FUNCTION_BLOCK A2X_PUBLISH_2 (* Publish both BOOLs of an A2X adapter to one or many SUBSCRIBE_2 Blocks, each buffered with an E_D_FF. Contract: garantiert seit v1.1 einen erzwungenen ersten Publish direkt nach INIT (OPC-UA-Knoten existiert sofort, auch ohne vorherige echte Wertaenderung am Adapter) - dieser erste Publish kann aber noch den Default-/Platzhalterwert des internen Latches enthalten statt des tatsaechlichen aktuellen Adapterwerts, bis die erste echte Aenderung eintrifft. Consumer, die auf den exakten Erstwert angewiesen sind, muessen das beruecksichtigen. Verhalten bei QI=FALSE (deaktivierter Publisher) verifiziert (FORTE-Quellcode, core/src/cominfra/commfb.cpp): weder beim INIT (Verbindung wird geschlossen statt geoeffnet) noch beim erzwungenen Erst-Publish (sendData() bricht vor dem Erreichen der Kommunikationsschicht ab) wird tatsaechlich etwas gesendet oder ein Knoten angelegt - das dabei ausgeloeste CNF/QO=FALSE/STATUS=Inhibited ist reine lokale Rueckmeldung, keine Netzwerkoperation, unbedenklich. Ein spaeterer QI-Wechsel FALSE->TRUE ohne erneutes INIT loest den erzwungenen Erst-Publish NICHT erneut aus. *)
  (* Standard: 61499-2; Description: Copyright (c) 2026 HR Agrartechnik GmbH This program and the accompanying materials are made available under the terms of the Eclipse Public License 2.0 which is available at https://www.eclipse.org/legal/epl-2.0/ SPDX-License-Identifier: EPL-2.0 *)
  (* Version 1.1, 2026-09-17, Franz Höpfinger, HR Agrartechnik GmbH, Erzwungener Erst-Publish nach INIT: PUBLISH_1/PUBLISH_2.INITO -> .REQ ergaenzt (Franz, gegen fehlende OPC-UA-Knoten wenn seit Power-On noch keine echte Wertaenderung stattfand, siehe BERICHT_2026-09-16_STG3_I1_I3_I4_I6_STALE_REMOTE_SUBSCRIBE.md Abschnitt 18-20) - garantiert einen unbedingten ersten Publish direkt nach der Initialisierung. *)
  (* Version 1.0, 2026-09-05, Franz Höpfinger, HR Agrartechnik GmbH, initial API and implementation and/or initial documentation *)
  PACKAGE adapter::net;
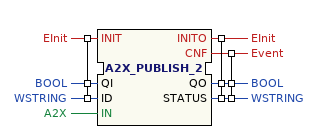
  EVENT_INPUT
    INIT : EInit WITH QI, ID; (* Initialization *)
  END_EVENT
  EVENT_OUTPUT
    INITO : EInit WITH QO, STATUS; (* Initialization Confirm *)
    CNF WITH QO, STATUS; (* Data was sent *)
  END_EVENT
  VAR_INPUT
    QI : BOOL;
    ID : WSTRING;
  END_VAR
  VAR_OUTPUT
    QO : BOOL;
    STATUS : WSTRING;
  END_VAR
  SOCKETS
    IN : adapter::types::unidirectional::A2X; (* UP/DOWN BOOLs to publish *)
  END_SOCKETS
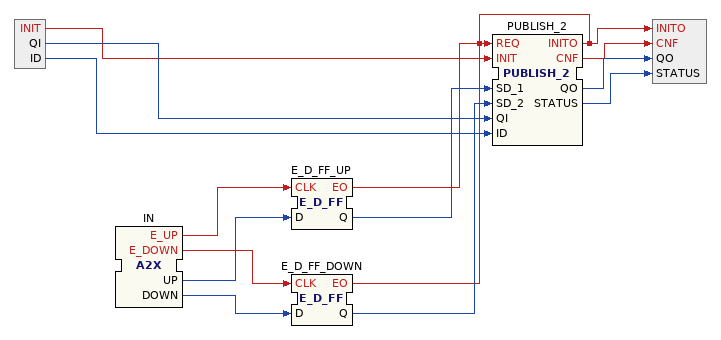
  FBS
    E_D_FF_UP : iec61499::events::E_D_FF;
    E_D_FF_DOWN : iec61499::events::E_D_FF;
    PUBLISH_2 : iec61499::net::PUBLISH_2;
  END_FBS
  EVENT_CONNECTIONS
    PUBLISH_2.INITO TO INITO;
    PUBLISH_2.CNF TO CNF;
    IN.E_UP TO E_D_FF_UP.CLK;
    IN.E_DOWN TO E_D_FF_DOWN.CLK;
    E_D_FF_UP.EO TO PUBLISH_2.REQ;
    E_D_FF_DOWN.EO TO PUBLISH_2.REQ;
    INIT TO PUBLISH_2.INIT;
    PUBLISH_2.INITO TO PUBLISH_2.REQ;
  END_CONNECTIONS
  DATA_CONNECTIONS
    PUBLISH_2.QO TO QO;
    PUBLISH_2.STATUS TO STATUS;
    IN.UP TO E_D_FF_UP.D;
    IN.DOWN TO E_D_FF_DOWN.D;
    E_D_FF_UP.Q TO PUBLISH_2.SD_1;
    E_D_FF_DOWN.Q TO PUBLISH_2.SD_2;
    QI TO PUBLISH_2.QI;
    ID TO PUBLISH_2.ID;
  END_CONNECTIONS
END_FUNCTION_BLOCK
